{attribute 'qualified_only'}
{attribute 'strict'}
TYPE Homing :
(
	IDLE,
	HOME_OUT,
	HOME_FINAL,
	STOP,
	SET,
	DONE,
	REDO
);
END_TYPE

(* stored: Version 1.1.0.1, ProductVersion 3.1.4024.11
   DUT Homing: Id {8cb9de35-a383-425e-8ca1-d663d47beaf0} *)
